{attribute addProperty BoxType "EP1816-0008-0016"}
{attribute addProperty Id "DO_Inputs_ChannelAT %I*ARRAY[0..1] OF DO_Inputs_Channel_9F71B9E2144180WcStateAT %I*WcState_98A4DF7520.250InfoDataAT %I*InfoData_BC63D37F80100"}
{attribute addProperty CRC "1461858632"}
{attribute addProperty SizeInBites "226"}
{attribute addProperty SizeInBytes "28.25"}
TYPE EP1816_5EE46DF6 :
STRUCT
	{attribute addProperty Name "DO_Inputs_Channel"}
	DO_Inputs_Channel : ARRAY[0..1] OF DO_Inputs_Channel_9F71B9E2;
	{attribute addProperty Name "WcState"}
	WcState : WcState_98A4DF75;
	{attribute addProperty Name "InfoData"}
	InfoData : InfoData_BC63D37F;
END_STRUCT
END_TYPE

(* stored: Version 1.2.0.0, ProductVersion 3.1.4024.9
   DUT EP1816_5EE46DF6: Id {11448e9b-8e68-43f9-8124-c57a1992bde1} *)
